// TIA Portal V16 export
// export: Created 2021-11-12T13:32:46.0888135Z, ExportSetting WithDefaults, DisplayName Totally Integrated Automation Portal, DisplayVersion V16 Update 3, DisplayName TIA Portal Version Control Interface, DisplayVersion V16 Update 2, DisplayName TIA Portal Openness, DisplayVersion V16 Update 3, DisplayName SINAMICS Startdrive Advanced, DisplayVersion V16 Update 5, DisplayName SINAMICS Startdrive G130, G150, S120, S150, SINAMICS MV, S210, DisplayVersion V16 Update 5, DisplayName SINAMICS Startdrive G110M, G120, G120C, G120D, G120P, G115D, DisplayVersion V16 Update 5, DisplayName STEP 7 Professional, DisplayVersion V16 Update 3, DisplayName STEP 7 Safety, DisplayVersion V16, DisplayName WinCC UA Professional, DisplayVersion V16 Update 3
DATA_BLOCK "HMI_CMD_Zone200"   // DB23
{ S7_Optimized_Access := 'TRUE'; DB_Accessible_From_OPC_UA := 'FALSE' }
VERSION : 0.1
// stored: AutoNumber true, DBAccessibleFromOPCUA false, IsOnlyStoredInLoadMemory false, IsRetainMemResEnabled false, IsWriteProtectedInAS false, MemoryReserve 100
   VAR
      Mode : "UDT_Zone_Command";   // Commands for zone 200
      Station210_Mode : "UDT_Station_Command";   // Commands for station 210
      Station220_Mode : "UDT_Station_Command";   // Commands for station 220
      Station230_Mode : "UDT_Station_Command";   // Commands for station 230
      Station2R1_Mode : "UDT_Station_Command";   // Commands for station 2R1
      Station2R2_Mode : "UDT_Station_Command";   // Commands for station 2R2
      StationSCH1_Mode : "UDT_Station_Command";   // Commands for forging station SCH1
      StationBSN3_Mode { S7_SetPoint := 'True'} : "UDT_Station_Command";   // Commands for furnace station BSN3
      StationsSum { S7_SetPoint := 'True'} : "UDT_StationsModesCmd";
      xxxxx___Alarms___xxxxx { S7_SetPoint := 'True'} : Byte;
      "200UF01-SF01" : "UDT_DI_Mon_Command";   // E-stop 200UF01-SF01
      "200QQ01_ES" { S7_SetPoint := 'True'} : "UDT_DI_Mon_Command";   // E-stop gate 200QQ01
      "200QQ02_ES" { S7_SetPoint := 'True'} : "UDT_DI_Mon_Command";   // E-stop gate 200QQ02
      "200QQ03_ES" { S7_SetPoint := 'True'} : "UDT_DI_Mon_Command";   // E-stop gate 200QQ03
      "200QQ04_ES" { S7_SetPoint := 'True'} : "UDT_DI_Mon_Command";   // E-stop gate 200QQ04
      "200QQ05_ES" { S7_SetPoint := 'True'} : "UDT_DI_Mon_Command";   // E-stop gate 200QQ05
      "200RU01-KF01" { S7_SetPoint := 'True'} : "UDT_DI_Mon_Command";   // gate module 200RU01-KF01
      "200RU01-KF02" { S7_SetPoint := 'True'} : "UDT_DI_Mon_Command";   // gate module 200RU01-KF02
      "200RU01-KF03" { S7_SetPoint := 'True'} : "UDT_DI_Mon_Command";   // gate module 200RU01-KF03
      "200RU01-KF04" { S7_SetPoint := 'True'} : "UDT_DI_Mon_Command";   // gate module 200RU01-KF04
   END_VAR
BEGIN
END_DATA_BLOCK
